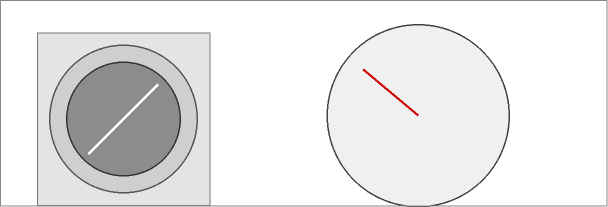
VISUALIZATION Visu_FC1_Test  // 608x207
    Group (37,24 571x183)
        Meter180 (191,0 380x183), value: GVL.geschrevenSnelheid, style: Meter-Meter180-Gray, scale format: %.1f, scale 0..200
        Potentiometer360 (0,7 173x176), variable: GVL.weegcelWaarde, style: Potentiometer-Potentiometer360-Gray, scale format: %.1f, scale 0..100
            p2431819421: Outside
END_VISUALIZATION

(* stored: Version 1.1.0.1, ProductVersion 3.1.4024.12
   Visu Visu_FC1_Test: Id {72a9fd95-2a00-4926-a32e-4e0c3c4e751a} *)
